INTERFACE RecipeStringValueType EXTENDS RecipeValue

METHOD ParseAndAssignValue
VAR_INPUT
END_VAR
END_METHOD

END_INTERFACE

(* stored: Version 1.1.0.1, ProductVersion 3.1.4024.15
   Itf RecipeStringValueType: Id {bc2726b3-c042-0db5-27a6-bc2ddbfc3f14}
   Method ParseAndAssignValue: Id {838f099f-ad86-04c7-241d-4a2cb15b2afb} *)
